PROGRAM MAIN
VAR
END_VAR

END_PROGRAM

(* stored: Version 1.1.0.1
   POU MAIN: Id {637085b5-c2e5-4e40-becc-298324a5f4a4} *)
